(* CoDeSys 2.3.9.47 project: gym_2016_12_27.pr6 *)
(* Libraries: PlcSystemBC.lb6 21.3.01 10:03:02, PlcHelperBC.lb6 7.5.01 10:03:00, TcAdsBC.lb6 5.7.02 10:03:02, standard.lib 5.6.98 10:03:02, TcBABasic.lib 22.7.15 14:46:14, TcPlcUtilitiesBC.lb6 13.5.05 10:19:40 *)

(* Global variable list: main *)
VAR_GLOBAL
	data3floor: ARRAY[0..100] OF BYTE;
	data3floor_prev :ARRAY[0..100] OF BYTE;

	ads_adr1: STRING:='10.0.5.61.1.1';
	ads_adr2: STRING:='10.0.5.62.1.1';
	ads_adr3: STRING:='10.0.5.63.1.1';

	write_ads: ADSWRITE;

	bDarkOutside		AT%MX0.0:BOOL;


	iHour			AT%MB4:BYTE;
	iMinute			AT%MB5:BYTE;
	lights			AT%MB6:DWORD;
	t_out			AT%MB10:INT;

	eib_gym01 						AT %MX100.0:	 BOOL;
	eib_gym02 						AT %MX100.1:	 BOOL;
	eib_training01 					AT %MX100.2:	 BOOL;
	eib_training02					AT %MX100.3:	 BOOL;
	eib_training03					AT %MX100.4:	 BOOL;
	eib_gym_stairs_bra				AT %MX100.5:	 BOOL;
	eib_pool_hall_spotlight			AT %MX100.6:	 BOOL;
	eib_pool_hall_LED				AT %MX100.7:	 BOOL;

	eib_pool_light 					AT %MX101.0:	 BOOL;
	eib_sphere_ceiling_light 			AT %MX101.1:	 BOOL;
	eib_sphere_light 				AT %MX101.2:	 BOOL;
	eib_gym_cinema_bra 			AT %MX101.3:	 BOOL;
	eib_gym_shower01_light			AT %MX101.4:	 BOOL;
	eib_gym_shower02_light			AT %MX101.5:	 BOOL;
	eib_gym_corridor_light			AT %MX101.6:	 BOOL;
	eib_gym_stairs_light 				AT %MX101.7:	 BOOL;

	eib_gym_WC_light 				AT %MX102.0:	 BOOL;
	eib_cinema_temporary_light		AT %MX102.1:	 BOOL;
END_VAR

(* POU MAIN, ST *)
PROGRAM MAIN
VAR
	i,j:INT;
	write:BOOL;
	heartBeat: TP;
END_VAR
heartBeat(IN:= NOT heartBeat.Q, PT:=t#5s);
Light;
write_data3floor;
(*ADS_Communication;*)
END_PROGRAM
ACTION write_data3floor:
	data3floor[0].0:= gym01_light ;
	data3floor[0].1:= gym02_light;
	data3floor[0].2:= training01_light;
	data3floor[0].3:= training02_light;
	data3floor[0].4:= training03_light;
	data3floor[0].5:= gym_stairs_bra_left;
	data3floor[0].6:= pool_hall_spotlight;
	data3floor[0].7:= pool_hall_LED;

	data3floor[1].0:= pool_light;
	data3floor[1].1:= sphere_ceiling_light;
	data3floor[1].2:= sphere_light01;
	data3floor[1].3:= gym_cinema_bra;
	data3floor[1].4:= gym_shower01_light;
	data3floor[1].5:= gym_shower02_light;
	data3floor[1].6:= gym_WC_corridor;
	data3floor[1].7:= gym_stairs_light;

	data3floor[2].0:= gym_WC_light;



FOR i:=0 TO (SIZEOF(data3floor))-1 DO
	IF data3floor[i]<>data3floor_prev[i]  THEN
		write:=TRUE;
		EXIT;
	ELSE
		write:=FALSE;
	END_IF
END_FOR


FOR j:=0 TO (SIZEOF(data3floor))-1 DO
	data3floor_prev[j]:=data3floor[j];
END_FOR
END_ACTION

(* POU Light, CFC *)
PROGRAM Light
VAR
	fb_gym01_light			: FB_Light;
	fb_gym02_light			: FB_Light;
	fb_training01_light		: FB_Light;
	fb_training02_light		: FB_Light;
	fb_training03_light		: FB_Light;
	fb_gym_stairs_bra		: FB_Light;
	fb_pool_hall_spotlight	: FB_Light;
	fb_pool_hall_LED		: FB_Light;
	fb_pool_light			: FB_Light;
	fb_sphere_ceiling_light	: FB_Light;
	fb_sphere_light			: FB_Light;
	fb_gym_cinema_bra		: FB_Light;
	fb_gym_shower01_light	: FB_Light;
	fb_gym_shower02_light	: FB_Light;
	fb_gym_corridor_light	: FB_Light;
	fb_gym_stairs_light		: FB_Light;
	fb_gym_WC_light		: FB_Light;


	fb_cinema_temporary_light	:FB_Light;

END_VAR
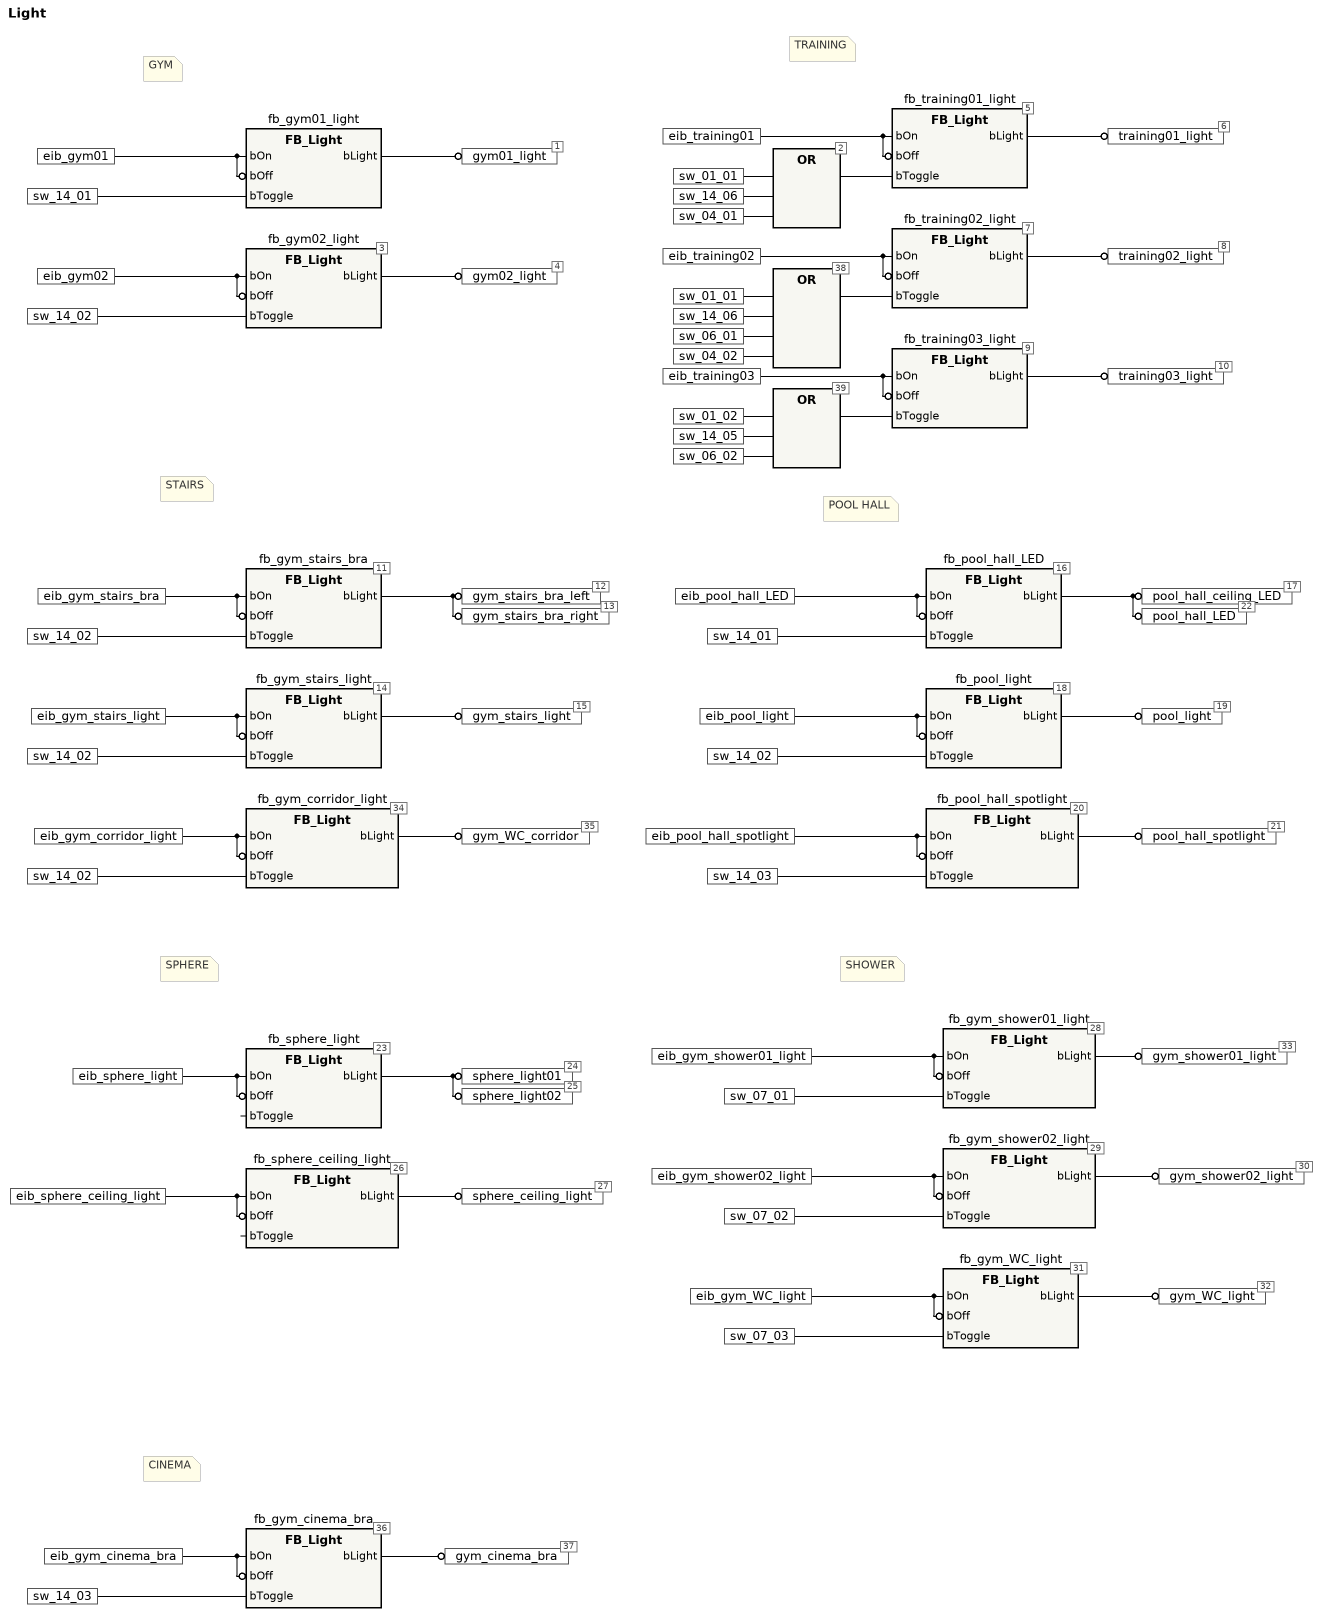
_CFC_ (* Continuous Function Chart, elements in execution order *)
(* GYM *)
#0 fb_gym01_light:FB_Light(bOn: eib_gym01, bOff: NOT eib_gym01, bToggle: sw_14_01)
#1 gym01_light <= NOT #0.bLight
#2 OR(sw_01_01, sw_14_06, sw_04_01)
#3 fb_gym02_light:FB_Light(bOn: eib_gym02, bOff: NOT eib_gym02, bToggle: sw_14_02)
#4 gym02_light <= NOT #3.bLight
(* TRAINING *)
(* STAIRS *)
#5 fb_training01_light:FB_Light(bOn: eib_training01, bOff: NOT eib_training01, bToggle: #2)
#6 training01_light <= NOT #5.bLight
#7 fb_training02_light:FB_Light(bOn: eib_training02, bOff: NOT eib_training02, bToggle: #38)
#8 training02_light <= NOT #7.bLight
#9 fb_training03_light:FB_Light(bOn: eib_training03, bOff: NOT eib_training03, bToggle: #39)
#10 training03_light <= NOT #9.bLight
#11 fb_gym_stairs_bra:FB_Light(bOn: eib_gym_stairs_bra, bOff: NOT eib_gym_stairs_bra, bToggle: sw_14_02)
#12 gym_stairs_bra_left <= NOT #11.bLight
#13 gym_stairs_bra_right <= NOT #11.bLight
#14 fb_gym_stairs_light:FB_Light(bOn: eib_gym_stairs_light, bOff: NOT eib_gym_stairs_light, bToggle: sw_14_02)
#15 gym_stairs_light <= NOT #14.bLight
(* POOL HALL *)
#16 fb_pool_hall_LED:FB_Light(bOn: eib_pool_hall_LED, bOff: NOT eib_pool_hall_LED, bToggle: sw_14_01)
#17 pool_hall_ceiling_LED <= NOT #16.bLight
#18 fb_pool_light:FB_Light(bOn: eib_pool_light, bOff: NOT eib_pool_light, bToggle: sw_14_02)
#19 pool_light <= NOT #18.bLight
#20 fb_pool_hall_spotlight:FB_Light(bOn: eib_pool_hall_spotlight, bOff: NOT eib_pool_hall_spotlight, bToggle: sw_14_03)
#21 pool_hall_spotlight <= NOT #20.bLight
#22 pool_hall_LED <= NOT #16.bLight
(* SPHERE *)
#23 fb_sphere_light:FB_Light(bOn: eib_sphere_light, bOff: NOT eib_sphere_light, bToggle: -)
#24 sphere_light01 <= NOT #23.bLight
#25 sphere_light02 <= NOT #23.bLight
#26 fb_sphere_ceiling_light:FB_Light(bOn: eib_sphere_ceiling_light, bOff: NOT eib_sphere_ceiling_light, bToggle: -)
#27 sphere_ceiling_light <= NOT #26.bLight
(* SHOWER *)
#28 fb_gym_shower01_light:FB_Light(bOn: eib_gym_shower01_light, bOff: NOT eib_gym_shower01_light, bToggle: sw_07_01)
#29 fb_gym_shower02_light:FB_Light(bOn: eib_gym_shower02_light, bOff: NOT eib_gym_shower02_light, bToggle: sw_07_02)
#30 gym_shower02_light <= NOT #29.bLight
#31 fb_gym_WC_light:FB_Light(bOn: eib_gym_WC_light, bOff: NOT eib_gym_WC_light, bToggle: sw_07_03)
#32 gym_WC_light <= NOT #31.bLight
#33 gym_shower01_light <= NOT #28.bLight
#34 fb_gym_corridor_light:FB_Light(bOn: eib_gym_corridor_light, bOff: NOT eib_gym_corridor_light, bToggle: sw_14_02)
#35 gym_WC_corridor <= NOT #34.bLight
(* CINEMA *)
#36 fb_gym_cinema_bra:FB_Light(bOn: eib_gym_cinema_bra, bOff: NOT eib_gym_cinema_bra, bToggle: sw_14_03)
#37 gym_cinema_bra <= NOT #36.bLight
#38 OR(sw_01_01, sw_14_06, sw_06_01, sw_04_02)
#39 OR(sw_01_02, sw_14_05, sw_06_02)
_END_CFC_
END_PROGRAM

(* POU ADS_Communication, CFC *)
PROGRAM ADS_Communication
VAR
	fb_floor3ADSwrite: ADSWRITE;


	counter_error,counter_busy: CTU;
END_VAR
VAR (* helpers for the ST form of the networks *)
	_t21 : DWORD;
	_t23 : DWORD;
	_t42 : BOOL;
END_VAR
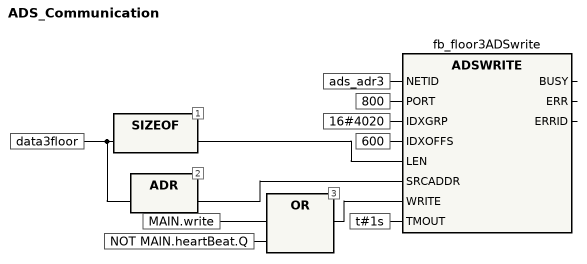
_CFC_ (* Continuous Function Chart, elements in execution order *)
#0 fb_floor3ADSwrite:ADSWRITE(NETID: ads_adr3, PORT: 800, IDXGRP: 16#4020, IDXOFFS: 600, LEN: #1, SRCADDR: #2, WRITE: #3, TMOUT: t#1s)
#1 SIZEOF(data3floor)
#2 ADR(data3floor)
#3 OR(MAIN.write, NOT MAIN.heartBeat.Q)
_END_CFC_
(* the same logic as Structured Text *)
fb_floor3ADSwrite(NETID := ads_adr3, PORT := 800, IDXGRP := 16#4020, IDXOFFS := 600, LEN := _t21, SRCADDR := _t23, WRITE := _t42, TMOUT := t#1s);
_t21 := SIZEOF(data3floor);
_t23 := ADR(data3floor);
_t42 := MAIN.write OR NOT MAIN.heartBeat.Q;
END_PROGRAM
